FUNCTION ElevatorFunction : BOOL

VAR_INPUT
	bCheckClass 	: BOOL;
END_VAR

VAR
	bMyDecision : BOOL;
END_VAR

IF bCheckClass THEN
	ElevatorFunction := TRUE;
ELSE
	ElevatorFunction := FALSE;
END_IF

END_FUNCTION

(* stored: Version 1.1.0.1, ProductVersion 3.1.4024.12
   POU ElevatorFunction: Id {c8d8a544-3236-4d33-bbe5-b48a60f9b991}, SpecialFunc None *)
